(* Logix 5000 project; controller Kollmeyer_LiveDemo_TBENLX8IOL_TBIL vendor 1 type 14 code 176 rev 32.11; software revision 32.00; part 8 of 9 *)
(* IOL_WriteData, continued *)

ROUTINE Prescan   (* ladder *)
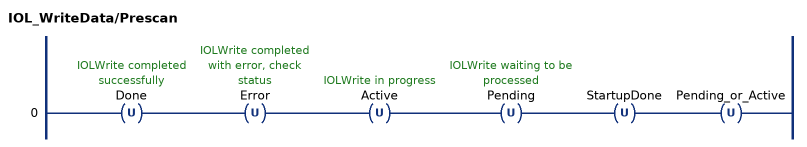
   0: OTU(Done)OTU(Error)OTU(Active)OTU(Pending)OTU(StartupDone)OTU(Pending_or_Active);
END_ROUTINE
END_ADD_ON_INSTRUCTION

ADD_ON_INSTRUCTION IOL_WriteString   (* revision 2.5 Support TBIP, ExecutePrescan, ExecuteEnableInFalse *)
// Revision note:
// V1_0 Initial Release
// V1_1 Documentation Update
// V1_3 Added multiple EIP node support
// V2_5 Support TBIP
// Help:
// IOL_WriteString - used with Turck BL20, BL67, BLC and TBEN IOLink masters to write string data to IOLink devices.  Use in conjuction with IOLService AOI which processes all IOL read and write requests.
// Status	Description
// 0	Operation completed successfully
// 	Status = 100 - 102, Ethernet IP MSG instruction errors - check communication parameters
// 100	IOL_SendMSG completed with error, check communication parameters
// 101	IOL_RecevieMSG completed with error, check communication parameters
// 110	IOL_Service Retry Limit exceeded
// 111	Slot specified not an IOLink master
// 	Status = 1000 to 1255, no response from device, connection error
// 1016	Device not connected or Port not configured as IOLink port
// 	Status = 2000 to 2255,  device response indicates error
// 2000	Device error, no details
// 2017	Device error, Index not available
// 2018	Device error, Subindex not available
// 2032	Device error, Service temporarily not available
// 2033	Device error, Service temporarily not available - local control
// 2034	Device error, Service temporarily not available - device control
// 2035	Device error, Index not writeable
// 2048	Device error, Parameter value out of range
// 2049	Device error, Parameter value above limit
// 2050	Device error, Parameter value below limit
// 2051	Device error, Parameter value length overrun (check IOLWrite precision/string length)
// 2052	Device error, Parameter value length underrun (check IOLWrite precision/string length)
// 2053	Device error, Function not available
// 2054	Device error, Function temporarily not available
// 2064	Device error, Parameter set invalid
// 2065	Device error, Inconsistent parameter set
// 2130	Device error, Application not ready
// 	Status = 3000 to 3255,   device response indicates vendor specific error
// 3000	Vendor specific error, no details
// 3001	Vendor specific error, vendor specific error number
// 3255	Vendor specific error, vendor specific error number
// 	Status = 7000 to 7255,  IOL-M Error Codes
// 7000	Unexpected write request instead of read request
// 7001	Decode error
// 7002	Port occupied by another task
// 	Status = 8000 to 8255,  IOL-M Error Codes
// 8000	Timeout when IOL-Ds or IOL-M ports are busy
// 8001	IOL Index out of range
// 8002	Port address greater than maximum
// 8003	Port function not supported
VAR_OUTPUT
   Done : BOOL; {access Read Only, visible}   // IOLWrite completed successfully
   Error : BOOL; {access Read Only, visible}   // IOLWrite completed with error, check status
   Pending : BOOL; {access Read Only, visible}   // IOLWrite waiting to be processed
   Active : BOOL; {access Read Only, visible}   // IOLWrite in progress
END_VAR
VAR_IN_OUT
   IOLData : Turck_IOL_CommonData; {required}   // Shared IOL Data Area - must be identical on all requests
END_VAR
VAR_OUTPUT
   DoneCount : DINT; {visible}   // Number of operations completed successfully
   ErrorCount : DINT; {access Read Only, visible}   // Number of operations competed with error
   Status : INT; {access Read Only, visible}   // Status of last IOLWrite
END_VAR
VAR_INPUT
   Write : BOOL;   // Rising edge triggers IOLink Write
   Slot : INT; {visible}   // IOLink Master slot number
   Port : INT; {visible}   // IOLink Master Port number, 1,2,3 or 4
   Index : INT; {visible}   // IOL Index number
   SubIndex : INT; {visible}   // IOL Subindex number
END_VAR
VAR_IN_OUT
   StringData : SINT[82]; {required}   // String data to write to IOLink device
END_VAR
VAR_INPUT
   StringLength : DINT; {access Read Only, required}   // Length of string data to write to IOLink device
END_VAR
VAR
   MyHandle : INT;
   StartupDone : BOOL; {access None}
   Pending_or_Active : BOOL; {access None}
   Write_ONS : BOOL; {access None}
   StartupCount : DINT; {access None}
   WriteRequest : BOOL; {access None}
END_VAR

ROUTINE EnableInFalse   (* ladder *)
END_ROUTINE

ROUTINE Logic   (* ladder *)
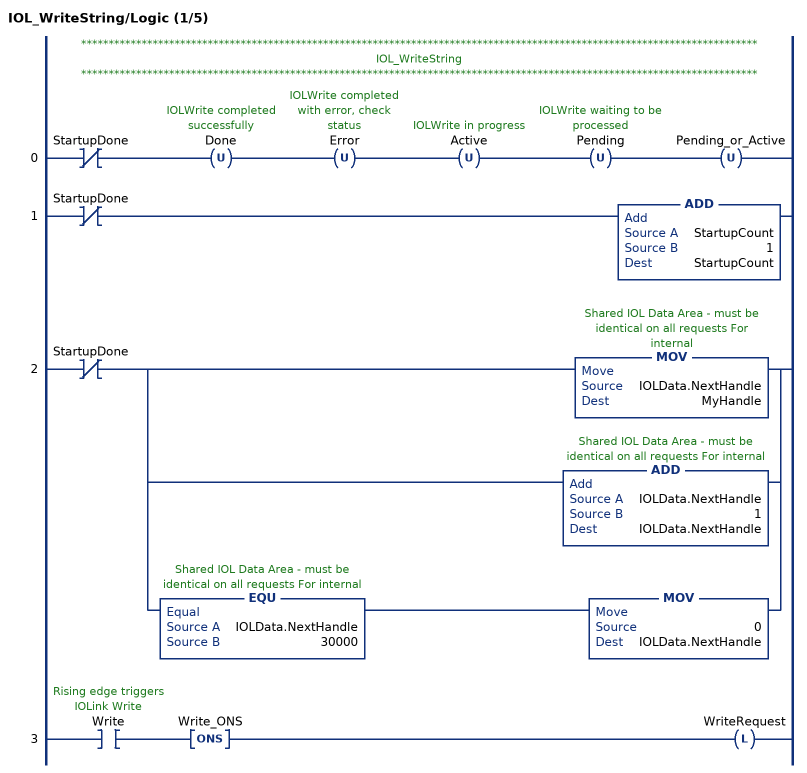
   // ***************************************************************************************************************************
   // IOL_WriteString
   // ***************************************************************************************************************************
   0: XIO(StartupDone)OTU(Done)OTU(Error)OTU(Active)OTU(Pending)OTU(Pending_or_Active);
   1: XIO(StartupDone)ADD(StartupCount,1,StartupCount);
   2: XIO(StartupDone)[MOV(IOLData.NextHandle,MyHandle) ,ADD(IOLData.NextHandle,1,IOLData.NextHandle) ,EQU(IOLData.NextHandle,30000) MOV(0,IOLData.NextHandle) ];
   3: XIC(Write)ONS(Write_ONS)OTL(WriteRequest);
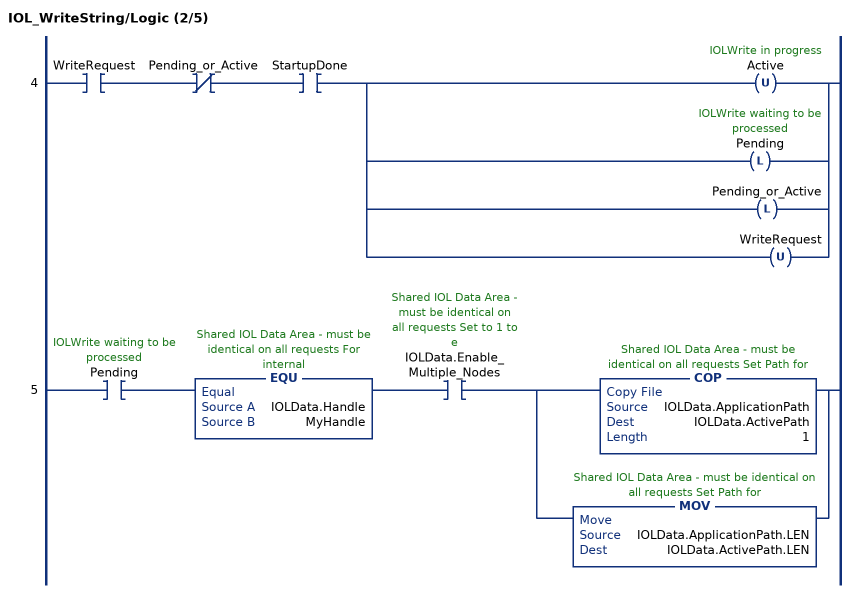
   4: XIC(WriteRequest)XIO(Pending_or_Active)XIC(StartupDone)[OTU(Active) ,OTL(Pending) ,OTL(Pending_or_Active) ,OTU(WriteRequest) ];
   5: XIC(Pending)EQU(IOLData.Handle,MyHandle)XIC(IOLData.Enable_Multiple_Nodes)[COP(IOLData.ApplicationPath,IOLData.ActivePath,1) ,MOV(IOLData.ApplicationPath.LEN,IOLData.ActivePath.LEN) ];
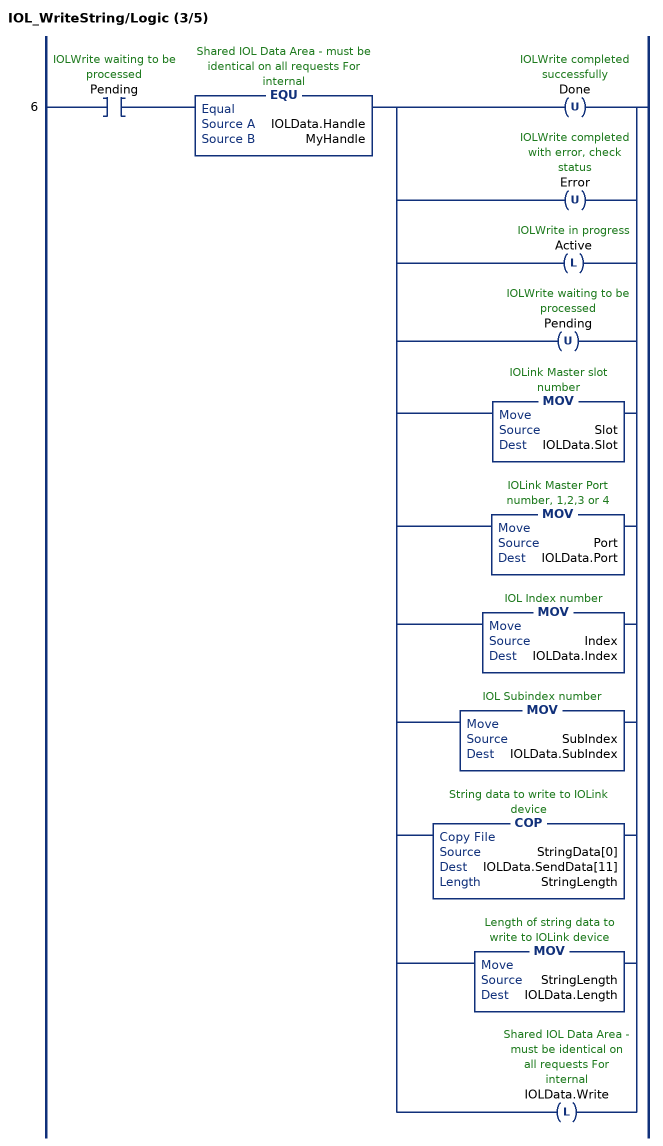
   6: XIC(Pending)EQU(IOLData.Handle,MyHandle)[OTU(Done) ,OTU(Error) ,OTL(Active) ,OTU(Pending) ,MOV(Slot,IOLData.Slot) ,MOV(Port,IOLData.Port) ,MOV(Index,IOLData.Index) ,MOV(SubIndex,IOLData.SubIndex) ,COP(StringData[0],IOLData.SendData[11],StringLength) ,MOV(StringLength,IOLData.Length) ,OTL(IOLData.Write) ];
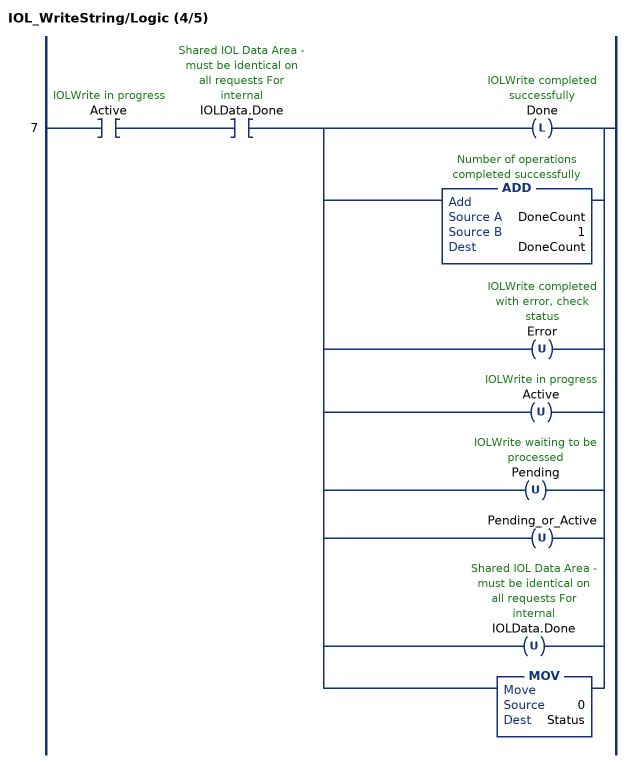
   7: XIC(Active)XIC(IOLData.Done)[OTL(Done) ,ADD(DoneCount,1,DoneCount) ,OTU(Error) ,OTU(Active) ,OTU(Pending) ,OTU(Pending_or_Active) ,OTU(IOLData.Done) ,MOV(0,Status) ];
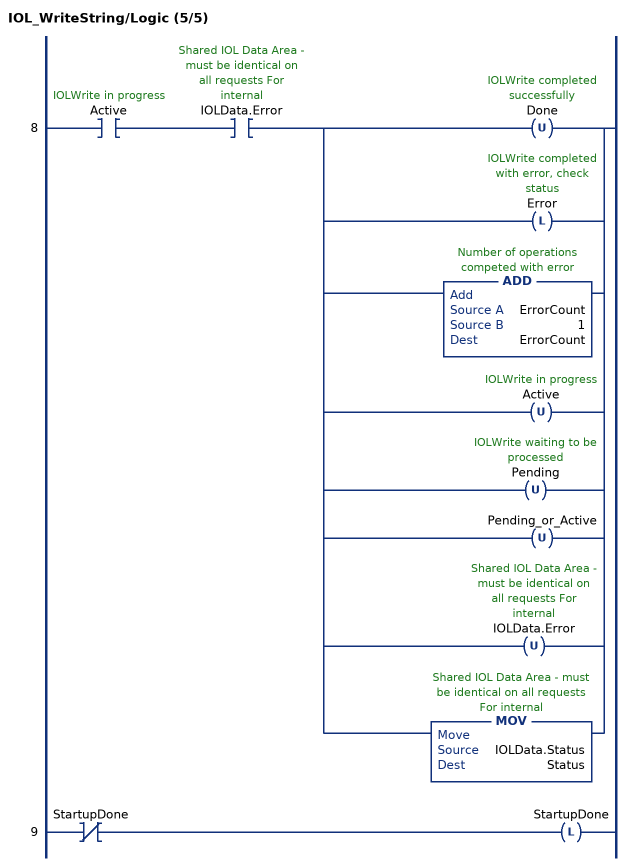
   8: XIC(Active)XIC(IOLData.Error)[OTU(Done) ,OTL(Error) ,ADD(ErrorCount,1,ErrorCount) ,OTU(Active) ,OTU(Pending) ,OTU(Pending_or_Active) ,OTU(IOLData.Error) ,MOV(IOLData.Status,Status) ];
   9: XIO(StartupDone)OTL(StartupDone);
END_ROUTINE

ROUTINE Prescan   (* ladder *)
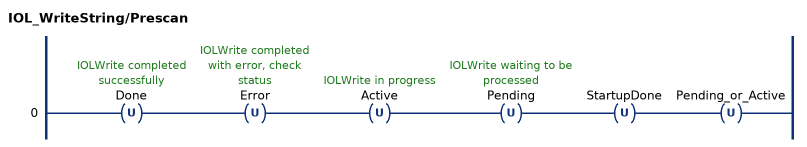
   0: OTU(Done)OTU(Error)OTU(Active)OTU(Pending)OTU(StartupDone)OTU(Pending_or_Active);
END_ROUTINE
END_ADD_ON_INSTRUCTION

ADD_ON_INSTRUCTION TBEN_L_8IOL_AOI   (* revision 0.1 Support TBIP, ExecutePrescan *)
// TBEN_L_8IOL AOI for managing all data to/from IOL blocks including process/acyclic data.
// Revision note:
// V0_1 Testing
// Help:
// IOL_Service - used with Turck BL20, BL67, BLC and TBEN IOLink masters to process requests from IOL_ReadString, IOL_WriteString, IOL_ReadData and IOL_WriteData AOI's.
// Status	Description
// 0	Operation completed successfully
// 	Status = 100 - 102, Ethernet IP MSG instruction errors - check communication parameters
// 100	IOL_SendMSG completed with error, check communication parameters
// 101	IOL_RecevieMSG completed with error, check communication parameters
// 110	IOL_Service Retry Limit exceeded
// 111	Slot specified not an IOLink master
// 	Status = 1000 to 1255, no response from device, connection error
// 1016	Device not connected or Port not configured as IOLink port
// 	Status = 2000 to 2255,  device response indicates error
// 2000	Device error, no details
// 2017	Device error, Index not available
// 2018	Device error, Subindex not available
// 2032	Device error, Service temporarily not available
// 2033	Device error, Service temporarily not available - local control
// 2034	Device error, Service temporarily not available - device control
// 2035	Device error, Index not writeable
// 2048	Device error, Parameter value out of range
// 2049	Device error, Parameter value above limit
// 2050	Device error, Parameter value below limit
// 2051	Device error, Parameter value length overrun (check IOLWrite precision/string length)
// 2052	Device error, Parameter value length underrun (check IOLWrite precision/string length)
// 2053	Device error, Function not available
// 2054	Device error, Function temporarily not available
// 2064	Device error, Parameter set invalid
// 2065	Device error, Inconsistent parameter set
// 2130	Device error, Application not ready
// 	Status = 3000 to 3255,   device response indicates vendor specific error
// 3000	Vendor specific error, no details
// 3001	Vendor specific error, vendor specific error number
// 3255	Vendor specific error, vendor specific error number
// 	Status = 7000 to 7255,  IOL-M Error Codes
// 7000	Unexpected write request instead of read request
// 7001	Decode error
// 7002	Port occupied by another task
// 	Status = 8000 to 8255,  IOL-M Error Codes
// 8000	Timeout when IOL-Ds or IOL-M ports are busy
// 8001	IOL Index out of range
// 8002	Port address greater than maximum
// 8003	Port function not supported
VAR_IN_OUT
   Process_Input_Data : Generic_173_Words; {required}
   Process_Output_Data : Generic_131_Words; {required}
   CommonData : Turck_IOL_CommonData; {required}
        .ReceiveData[2]   // KH changed from -9 (f7) to -4 (Fd)
        .SendData[1]   // For internal use to integrate IOLRead and IOLWrite with IOLService
   IOL_SendMSG : MESSAGE; {required}
   IOL_ReceiveMSG : MESSAGE; {required}
END_VAR
VAR_OUTPUT
   Port1_VID : DINT; {visible}
   Port1_DID : DINT; {visible}
   Port2_VID : DINT; {visible}
   Port2_DID : DINT; {visible}
   Port3_VID : DINT; {visible}
   Port3_DID : DINT; {visible}
   Port4_VID : DINT; {visible}
   Port4_DID : DINT; {visible}
   Port5_VID : DINT; {visible}
   Port5_DID : DINT; {visible}
   Port6_VID : DINT; {visible}
   Port6_DID : DINT; {visible}
   Port7_VID : DINT; {visible}
   Port7_DID : DINT; {visible}
   Port8_VID : DINT; {visible}
   Port8_DID : DINT; {visible}
   Port1_SN : DINT; {access Read Only}
   Port1_COMRev : DINT;
   Port1_ProcInLenght : DINT;
   Port1_ProcOutLenght : DINT;
   Port1_CycleTime : DINT;
   Port2_SN : DINT;
   Port2_COMRev : DINT;
   Port2_ProcInLenght : DINT;
   Port2_ProcOutLenght : DINT;
   Port2_CycleTime : DINT;
   Port3_SN : DINT;
   Port3_COMRev : DINT;
   Port3_ProcInLenght : DINT;
   Port3_ProcOutLenght : DINT;
   Port3_CycleTime : DINT;
   Port4_SN : DINT;
   Port4_COMRev : DINT;
   Port4_ProcInLenght : DINT;
   Port4_ProcOutLenght : DINT;
   Port4_CycleTime : DINT;
   Port5_SN : DINT;
   Port5_COMRev : DINT;
   Port5_ProcInLenght : DINT;
   Port5_ProcOutLenght : DINT;
   Port5_CycleTime : DINT;
   Port6_SN : DINT;
   Port6_COMRev : DINT;
   Port6_ProcInLenght : DINT;
   Port6_ProcOutLenght : DINT;
   Port6_CycleTime : DINT;
   Port7_SN : DINT;
   Port7_COMRev : DINT;
   Port7_ProcInLenght : DINT;
   Port7_ProcOutLenght : DINT;
   Port7_CycleTime : DINT;
   Port8_SN : DINT;
   Port8_COMRev : DINT;
   Port8_ProcInLenght : DINT;
   Port8_ProcOutLenght : DINT;
   Port8_CycleTime : DINT;
END_VAR
VAR
   IOLS1 : BOOL;
   IOLS2 : BOOL;
   IOLS3 : BOOL;
   IOLS4 : BOOL;
   IOLS5 : BOOL;
   IOLS6 : BOOL;
   IOLS7 : BOOL;
   IOLReadActive : BOOL;
   IOLWriteActive : BOOL;
   Retry : BOOL;
   RetryCount : DINT;
   IOL_SendMSG_Request : BOOL; {access None}
   IOL_ReceiveMSG_Request : BOOL; {access None}
   IOLS4_Bad : BOOL; {access None}
   IOL_S2_0_Count : DINT; {access None}
   IOL_S6_0_Count : DINT; {access None}
   Busy_Retry : BOOL; {access None}
   IOL_S2_0_Total : DINT; {access None}
   IOL_S3_Retry : DINT; {access None}
   IOL_S1_Count : DINT; {access None}
   IOL_S2_Count : DINT; {access None}
   IOL_S3_Count : DINT; {access None}
   IOL_S5_Count : DINT; {access None}
   IOL_S6_Count : DINT; {access None}
   ER1 : BOOL; {access None}
   ER2 : BOOL; {access None}
   IOL_S6_NotBusy_Count : DINT; {access None}
   RetryTotal : DINT; {access None}
   IOL_S4_Bad_Count : DINT; {access None}
   IOL_S2_Error_Count : DINT; {access None}
   IOL_Done_Count : DINT; {access None}
   IOL_Error_Count : DINT; {access None}
   IOLReset_ONS : BOOL; {access None}
   ABS_RD_11 : INT; {access None}
   ABS_RD_12 : INT; {access None}
   ABS_RD_13 : INT; {access None}
   IOL_SendMSG_DN : BOOL; {access None}
   IOL_ReceiveMSG_DN : BOOL; {access None}
   IOLS2A : BOOL; {access None}
   Generate_Status : BOOL; {access None}
   IOLS5A : BOOL; {access None}
   Busy_Response : BOOL; {access None}
   Done_Response : BOOL; {access None}
   IOL_S6_Done_Count : DINT; {access None}
   Wait : BOOL; {access None}
   IOL_S6_Busy_Count : DINT; {access None}
   PORT_DATA : SINT[230]; {access None}
   PORT_DATA_LENGHT : DINT; {access None}
   READ_PORT_DATA : IOL_ReadString := (Slot := 1, Index := -1, SubIndex := 68); {access None}
END_VAR

ROUTINE Logic   (* ladder *)
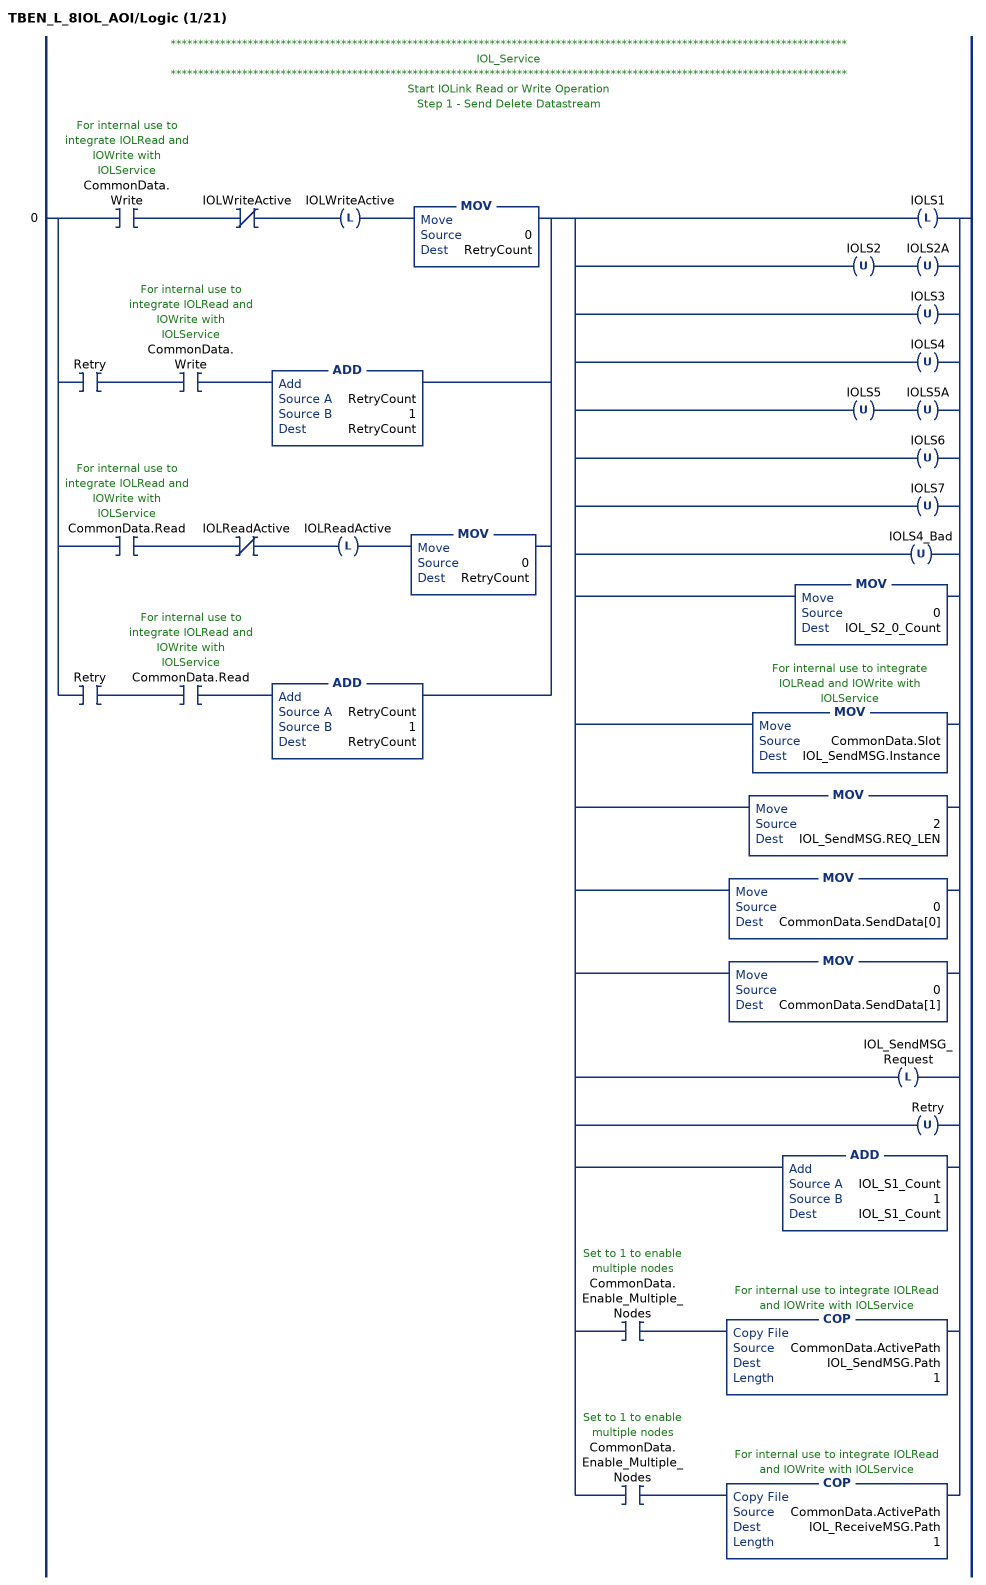
   // ***************************************************************************************************************************
   // IOL_Service
   // ***************************************************************************************************************************
   // Start IOLink Read or Write Operation
   // Step 1 - Send Delete Datastream
   0: [XIC(CommonData.Write) XIO(IOLWriteActive) OTL(IOLWriteActive) MOV(0,RetryCount) ,XIC(Retry) XIC(CommonData.Write) ADD(RetryCount,1,RetryCount) ,XIC(CommonData.Read) XIO(IOLReadActive) OTL(IOLReadActive) MOV(0,RetryCount) ,XIC(Retry) XIC(CommonData.Read) ADD(RetryCount,1,RetryCount) ][OTL(IOLS1) ,OTU(IOLS2) OTU(IOLS2A) ,OTU(IOLS3) ,OTU(IOLS4) ,OTU(IOLS5) OTU(IOLS5A) ,OTU(IOLS6) ,OTU(IOLS7) ,OTU(IOLS4_Bad) ,MOV(0,IOL_S2_0_Count) ,MOV(CommonData.Slot,IOL_SendMSG.Instance) ,MOV(2,IOL_SendMSG.REQ_LEN) ,MOV(0,CommonData.SendData[0]) ,MOV(0,CommonData.SendData[1]) ,OTL(IOL_SendMSG_Request) ,OTU(Retry) ,ADD(IOL_S1_Count,1,IOL_S1_Count) ,XIC(CommonData.Enable_Multiple_Nodes) COP(CommonData.ActivePath,IOL_SendMSG.Path,1) ,XIC(CommonData.Enable_Multiple_Nodes) COP(CommonData.ActivePath,IOL_ReceiveMSG.Path,1) ];
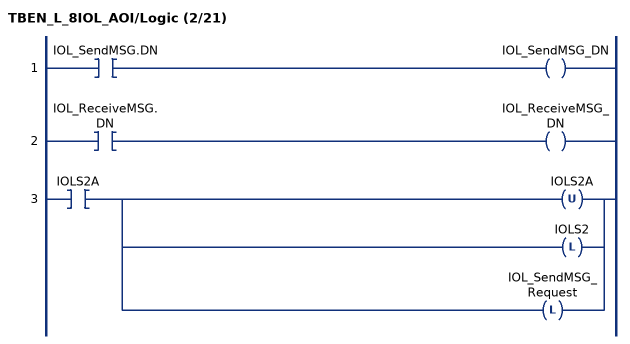
   1: XIC(IOL_SendMSG.DN)OTE(IOL_SendMSG_DN);
   2: XIC(IOL_ReceiveMSG.DN)OTE(IOL_ReceiveMSG_DN);
   3: XIC(IOLS2A)[OTU(IOLS2A) ,OTL(IOLS2) ,OTL(IOL_SendMSG_Request) ];
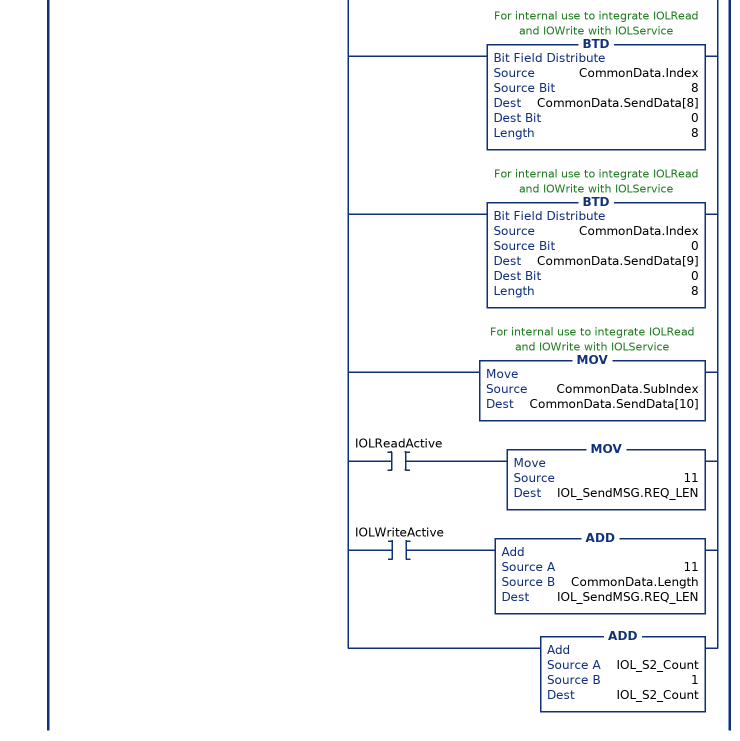
   // Step 1 - After Delete Stream sent then Send IOLink Read or Write Request
   4: XIC(IOLS1)XIC(IOL_SendMSG_DN)XIO(IOL_SendMSG_Request)[OTU(IOLS1) ,OTL(IOLS2A) ,MOV(CommonData.Slot,IOL_SendMSG.Instance) ,MOV(0,CommonData.SendData[0]) ,MOV(16#fc,CommonData.SendData[1]) ,MOV(16#11,CommonData.SendData[2]) ,MOV(16#08,CommonData.SendData[3]) ,MOV(CommonData.Port,CommonData.SendData[4]) ,MOV(16#fe,CommonData.SendData[5]) ,MOV(16#4a,CommonData.SendData[6]) ,XIC(IOLReadActive) MOV(16#03,CommonData.SendData[7]) ,XIC(IOLWriteActive) MOV(16#02,CommonData.SendData[7]) ,BTD(CommonData.Index,8,CommonData.SendData[8],0,8) ,BTD(CommonData.Index,0,CommonData.SendData[9],0,8) ,MOV(CommonData.SubIndex,CommonData.SendData[10]) ,XIC(IOLReadActive) MOV(11,IOL_SendMSG.REQ_LEN) ,XIC(IOLWriteActive) ADD(11,CommonData.Length,IOL_SendMSG.REQ_LEN) ,ADD(IOL_S2_Count,1,IOL_S2_Count) ];
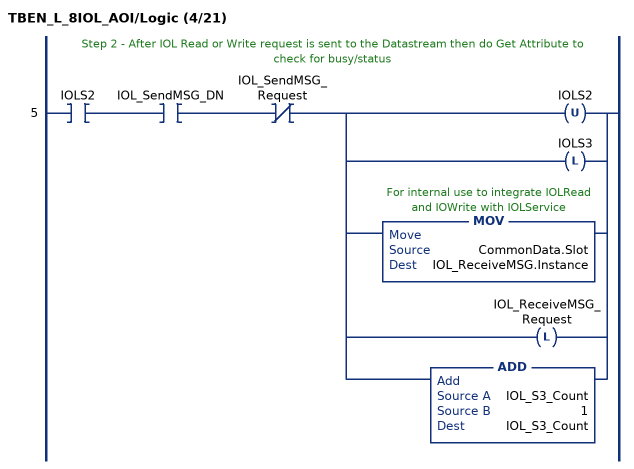
   // Step 2 - After IOL Read or Write request is sent to the Datastream then do Get Attribute to check for busy/status
   5: XIC(IOLS2)XIC(IOL_SendMSG_DN)XIO(IOL_SendMSG_Request)[OTU(IOLS2) ,OTL(IOLS3) ,MOV(CommonData.Slot,IOL_ReceiveMSG.Instance) ,OTL(IOL_ReceiveMSG_Request) ,ADD(IOL_S3_Count,1,IOL_S3_Count) ];
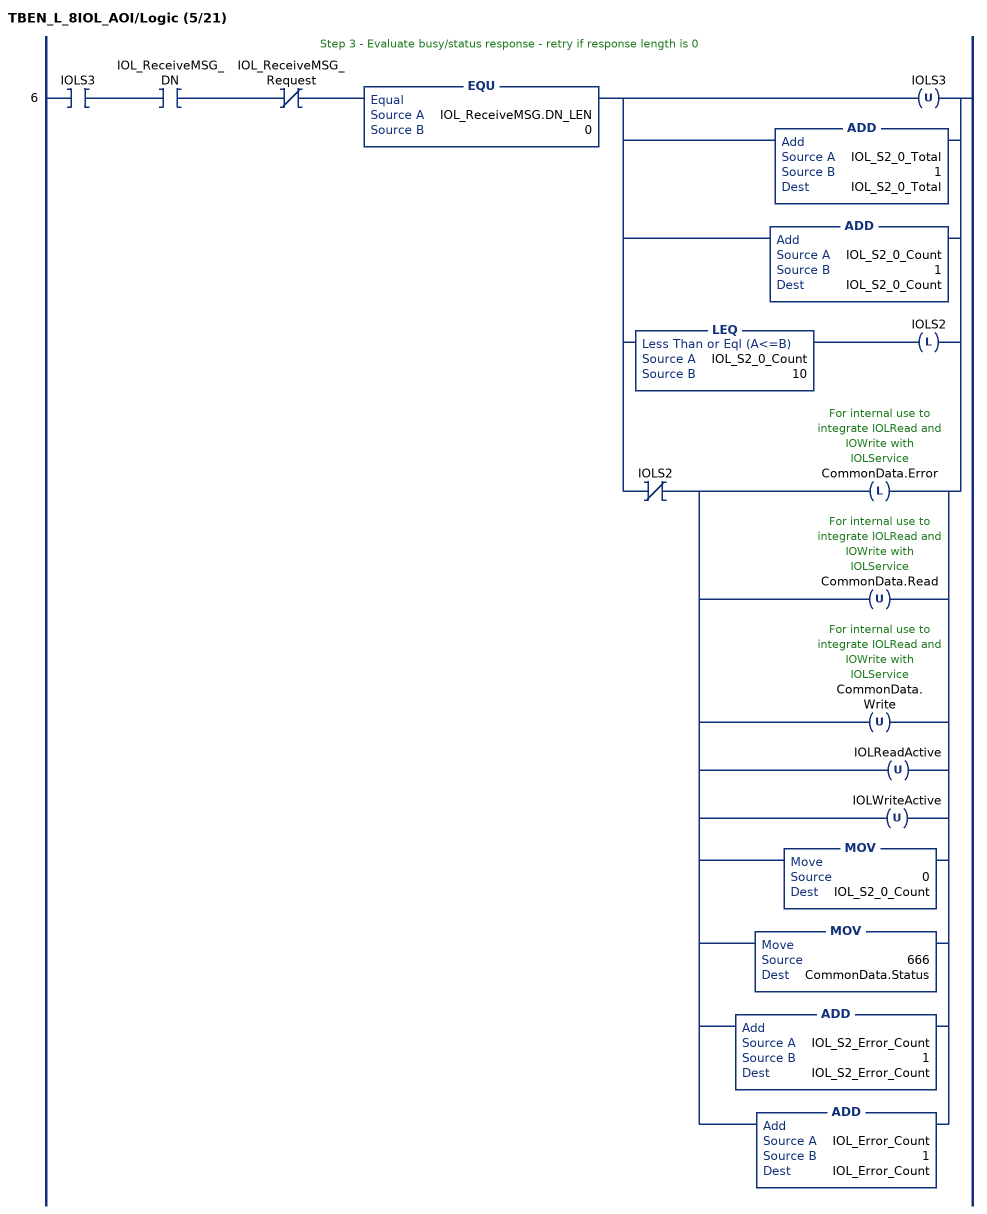
   // Step 3 - Evaluate busy/status response - retry if response length is 0
   6: XIC(IOLS3)XIC(IOL_ReceiveMSG_DN)XIO(IOL_ReceiveMSG_Request)EQU(IOL_ReceiveMSG.DN_LEN,0)[OTU(IOLS3) ,ADD(IOL_S2_0_Total,1,IOL_S2_0_Total) ,ADD(IOL_S2_0_Count,1,IOL_S2_0_Count) ,LEQ(IOL_S2_0_Count,10) OTL(IOLS2) ,XIO(IOLS2) [OTL(CommonData.Error) ,OTU(CommonData.Read) ,OTU(CommonData.Write) ,OTU(IOLReadActive) ,OTU(IOLWriteActive) ,MOV(0,IOL_S2_0_Count) ,MOV(666,CommonData.Status) ,ADD(IOL_S2_Error_Count,1,IOL_S2_Error_Count) ,ADD(IOL_Error_Count,1,IOL_Error_Count) ] ];
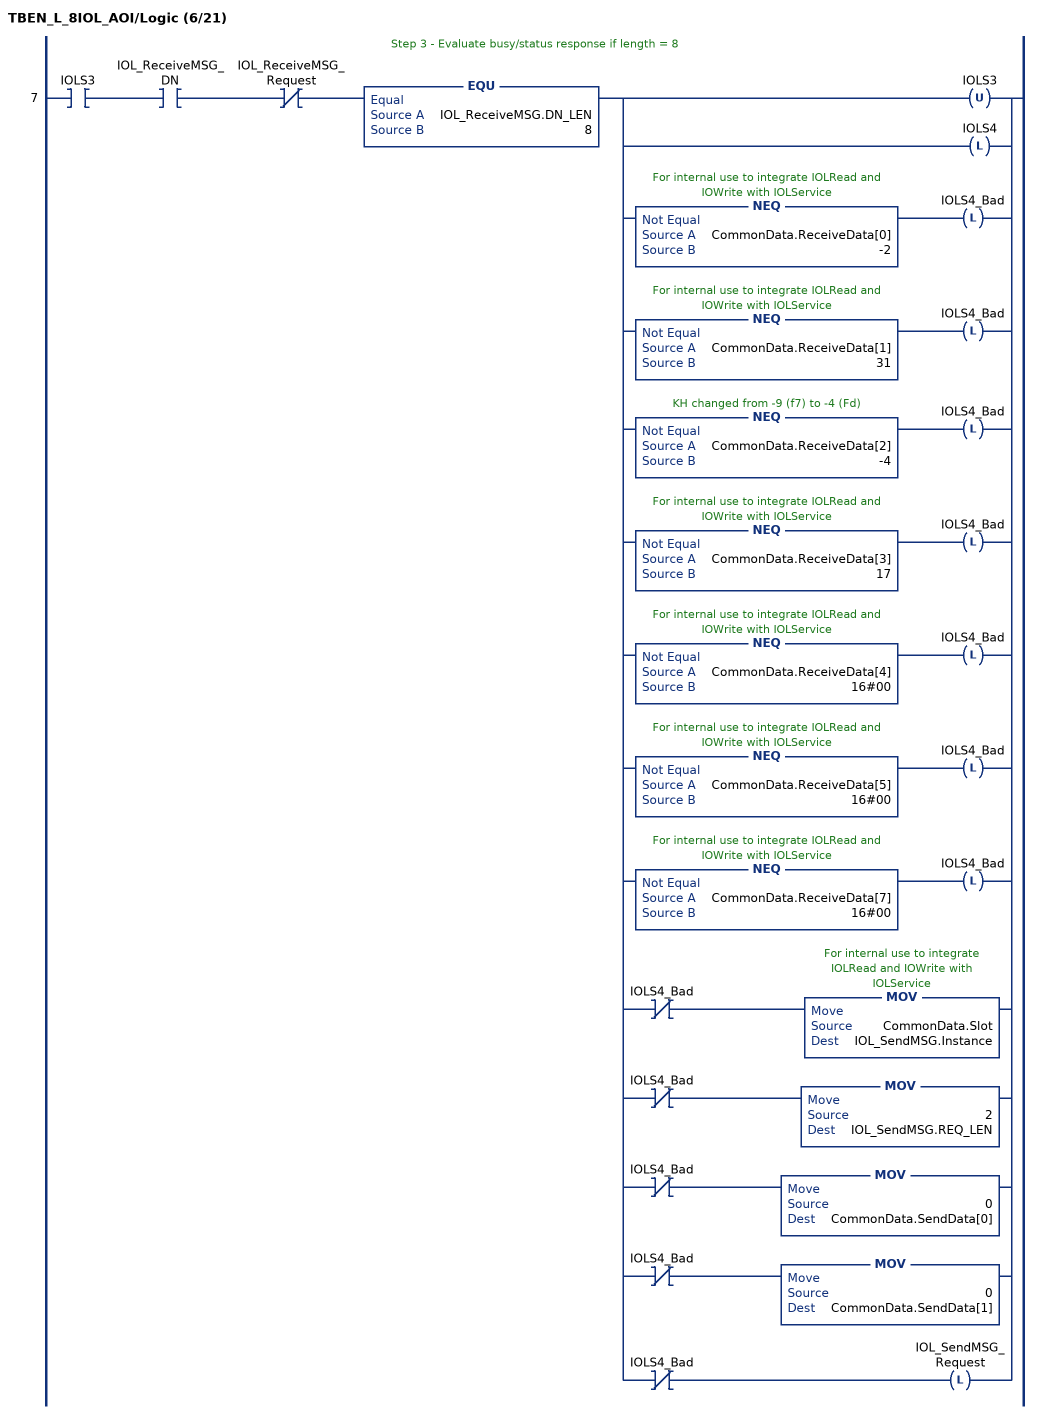
   // Step 3 - Evaluate busy/status response if length = 8
   7: XIC(IOLS3)XIC(IOL_ReceiveMSG_DN)XIO(IOL_ReceiveMSG_Request)EQU(IOL_ReceiveMSG.DN_LEN,8)[OTU(IOLS3) ,OTL(IOLS4) ,NEQ(CommonData.ReceiveData[0],-2) OTL(IOLS4_Bad) ,NEQ(CommonData.ReceiveData[1],31) OTL(IOLS4_Bad) ,NEQ(CommonData.ReceiveData[2],-4) OTL(IOLS4_Bad) ,NEQ(CommonData.ReceiveData[3],17) OTL(IOLS4_Bad) ,NEQ(CommonData.ReceiveData[4],16#00) OTL(IOLS4_Bad) ,NEQ(CommonData.ReceiveData[5],16#00) OTL(IOLS4_Bad) ,NEQ(CommonData.ReceiveData[7],16#00) OTL(IOLS4_Bad) ,XIO(IOLS4_Bad) MOV(CommonData.Slot,IOL_SendMSG.Instance) ,XIO(IOLS4_Bad) MOV(2,IOL_SendMSG.REQ_LEN) ,XIO(IOLS4_Bad) MOV(0,CommonData.SendData[0]) ,XIO(IOLS4_Bad) MOV(0,CommonData.SendData[1]) ,XIO(IOLS4_Bad) OTL(IOL_SendMSG_Request) ];
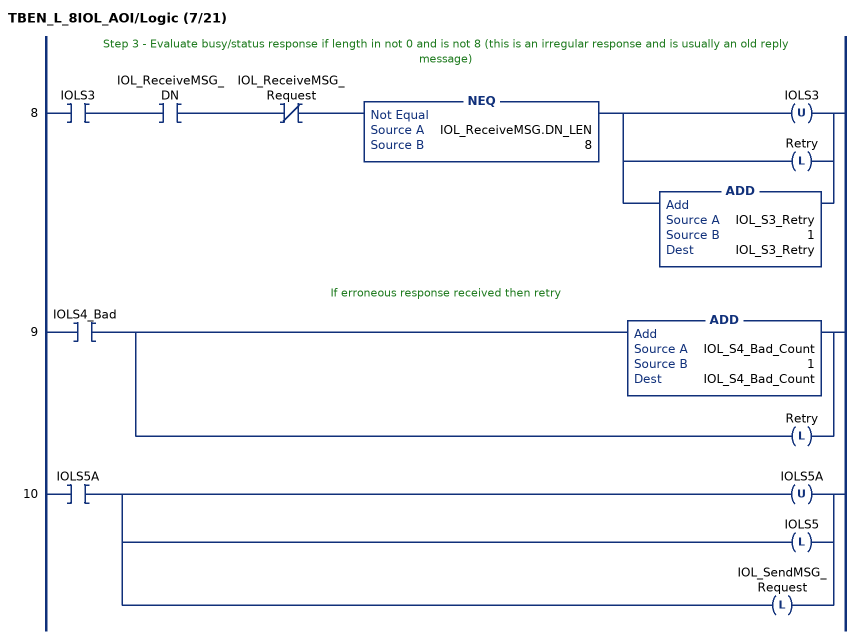
   // Step 3 - Evaluate busy/status response if length in not 0 and is not 8 (this is an irregular response and is usually an old reply message)
   8: XIC(IOLS3)XIC(IOL_ReceiveMSG_DN)XIO(IOL_ReceiveMSG_Request)NEQ(IOL_ReceiveMSG.DN_LEN,8)[OTU(IOLS3) ,OTL(Retry) ,ADD(IOL_S3_Retry,1,IOL_S3_Retry) ];
   // If erroneous response received then retry
   9: XIC(IOLS4_Bad)[ADD(IOL_S4_Bad_Count,1,IOL_S4_Bad_Count) ,OTL(Retry) ];
   10: XIC(IOLS5A)[OTU(IOLS5A) ,OTL(IOLS5) ,OTL(IOL_SendMSG_Request) ];
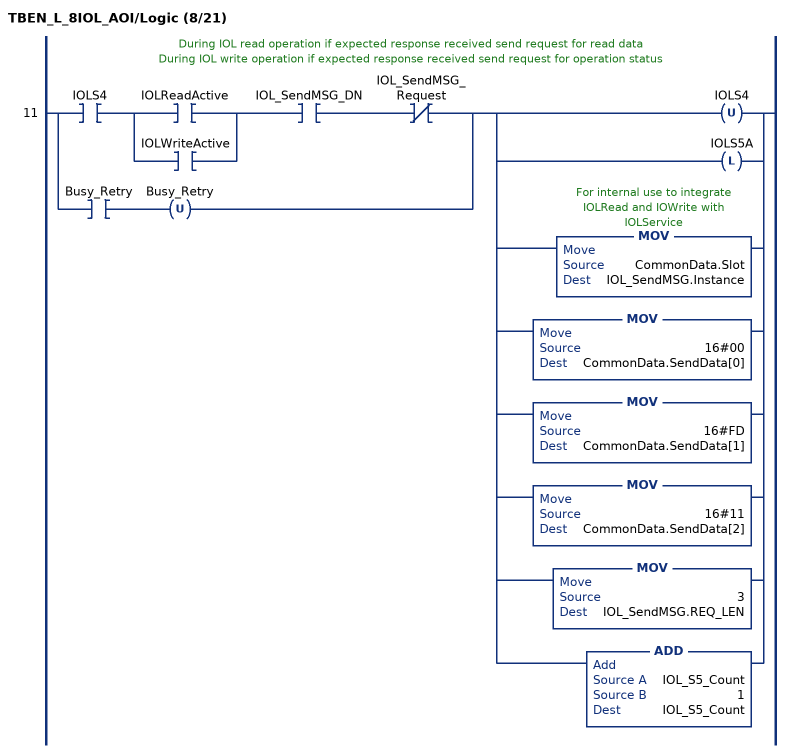
   // During IOL read operation if expected response received send request for read data
   // During IOL write operation if expected response received send request for operation status
   11: [XIC(IOLS4) [XIC(IOLReadActive) ,XIC(IOLWriteActive) ] XIC(IOL_SendMSG_DN) XIO(IOL_SendMSG_Request) ,XIC(Busy_Retry) OTU(Busy_Retry) ][OTU(IOLS4) ,OTL(IOLS5A) ,MOV(CommonData.Slot,IOL_SendMSG.Instance) ,MOV(16#00,CommonData.SendData[0]) ,MOV(16#FD,CommonData.SendData[1]) ,MOV(16#11,CommonData.SendData[2]) ,MOV(3,IOL_SendMSG.REQ_LEN) ,ADD(IOL_S5_Count,1,IOL_S5_Count) ];
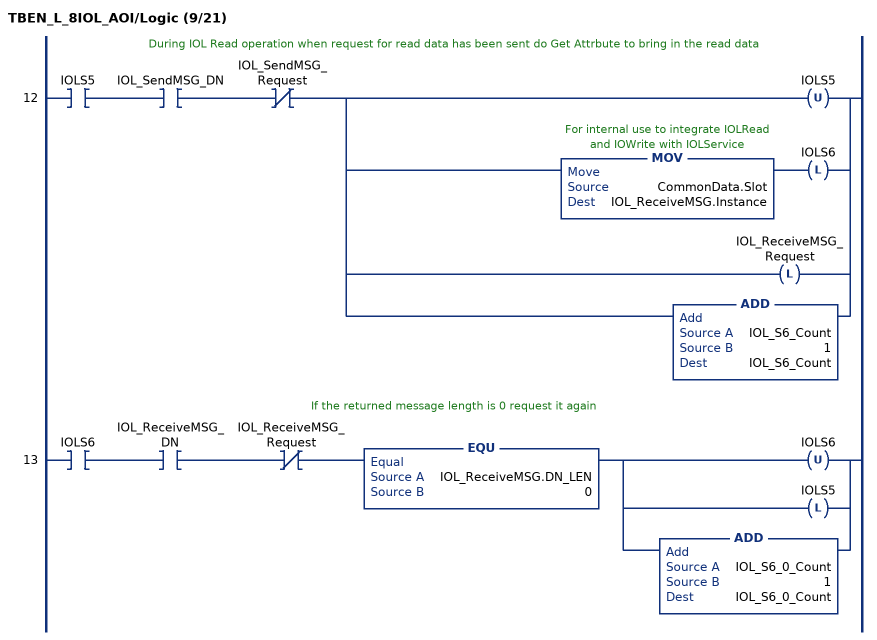
   // During IOL Read operation when request for read data has been sent do Get Attrbute to bring in the read data
   12: XIC(IOLS5)XIC(IOL_SendMSG_DN)XIO(IOL_SendMSG_Request)[OTU(IOLS5) ,MOV(CommonData.Slot,IOL_ReceiveMSG.Instance) OTL(IOLS6) ,OTL(IOL_ReceiveMSG_Request) ,ADD(IOL_S6_Count,1,IOL_S6_Count) ];
   // If the returned message length is 0 request it again
   13: XIC(IOLS6)XIC(IOL_ReceiveMSG_DN)XIO(IOL_ReceiveMSG_Request)EQU(IOL_ReceiveMSG.DN_LEN,0)[OTU(IOLS6) ,OTL(IOLS5) ,ADD(IOL_S6_0_Count,1,IOL_S6_0_Count) ];
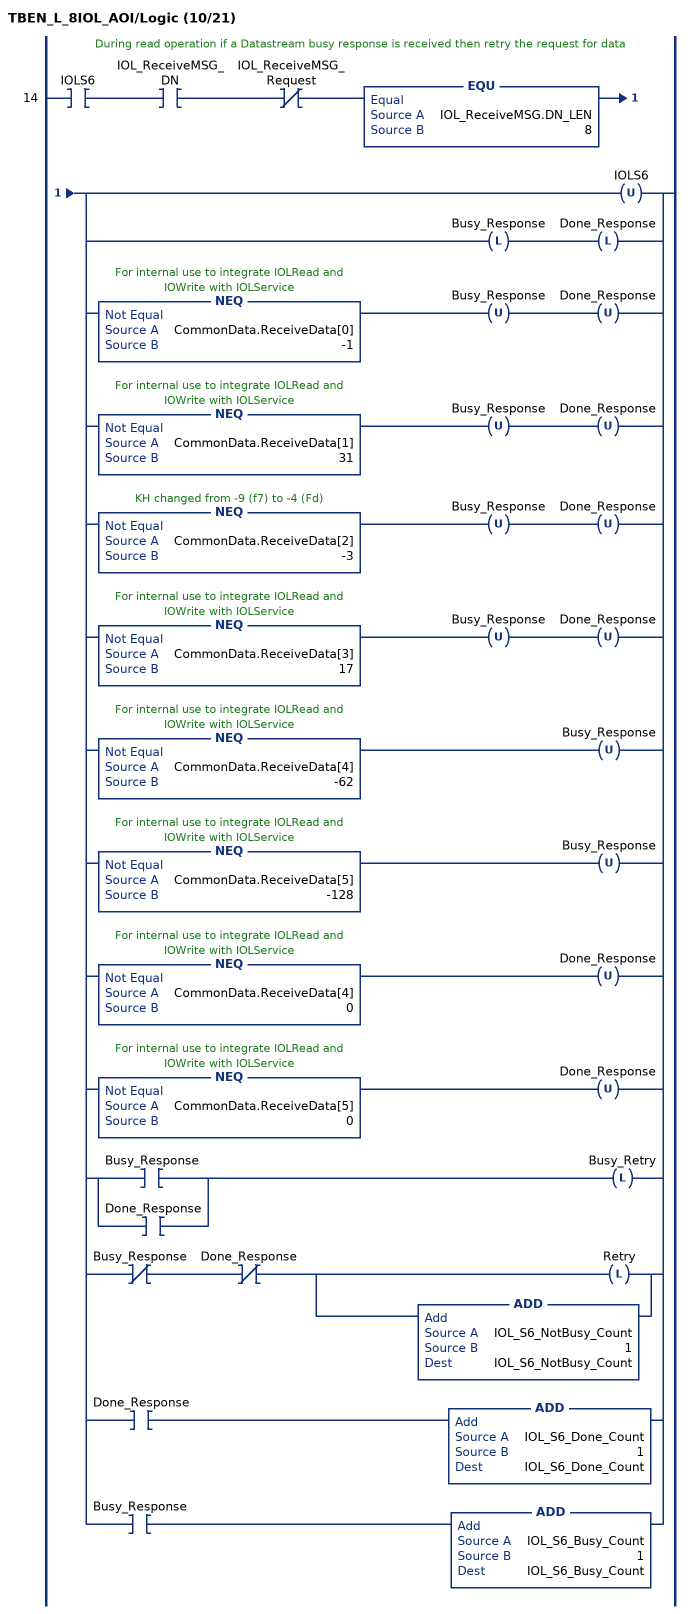
   // During read operation if a Datastream busy response is received then retry the request for data
   14: XIC(IOLS6)XIC(IOL_ReceiveMSG_DN)XIO(IOL_ReceiveMSG_Request)EQU(IOL_ReceiveMSG.DN_LEN,8)[OTU(IOLS6) ,OTL(Busy_Response) OTL(Done_Response) ,NEQ(CommonData.ReceiveData[0],-1) OTU(Busy_Response) OTU(Done_Response) ,NEQ(CommonData.ReceiveData[1],31) OTU(Busy_Response) OTU(Done_Response) ,NEQ(CommonData.ReceiveData[2],-3) OTU(Busy_Response) OTU(Done_Response) ,NEQ(CommonData.ReceiveData[3],17) OTU(Busy_Response) OTU(Done_Response) ,NEQ(CommonData.ReceiveData[4],-62) OTU(Busy_Response) ,NEQ(CommonData.ReceiveData[5],-128) OTU(Busy_Response) ,NEQ(CommonData.ReceiveData[4],0) OTU(Done_Response) ,NEQ(CommonData.ReceiveData[5],0) OTU(Done_Response) ,[XIC(Busy_Response) ,XIC(Done_Response) ] OTL(Busy_Retry) ,XIO(Busy_Response) XIO(Done_Response) [OTL(Retry) ,ADD(IOL_S6_NotBusy_Count,1,IOL_S6_NotBusy_Count) ] ,XIC(Done_Response) ADD(IOL_S6_Done_Count,1,IOL_S6_Done_Count) ,XIC(Busy_Response) ADD(IOL_S6_Busy_Count,1,IOL_S6_Busy_Count) ];
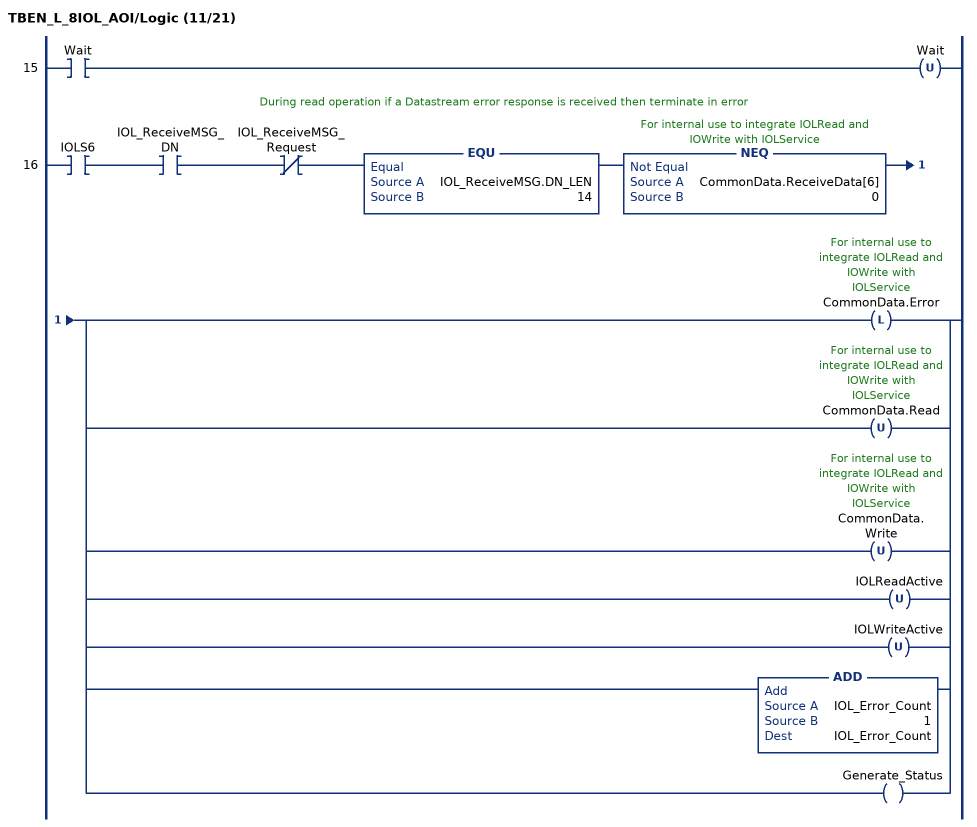
   15: XIC(Wait)OTU(Wait);
   // During read operation if a Datastream error response is received then terminate in error
   16: XIC(IOLS6)XIC(IOL_ReceiveMSG_DN)XIO(IOL_ReceiveMSG_Request)EQU(IOL_ReceiveMSG.DN_LEN,14)NEQ(CommonData.ReceiveData[6],0)[OTL(CommonData.Error) ,OTU(CommonData.Read) ,OTU(CommonData.Write) ,OTU(IOLReadActive) ,OTU(IOLWriteActive) ,ADD(IOL_Error_Count,1,IOL_Error_Count) ,OTE(Generate_Status) ];
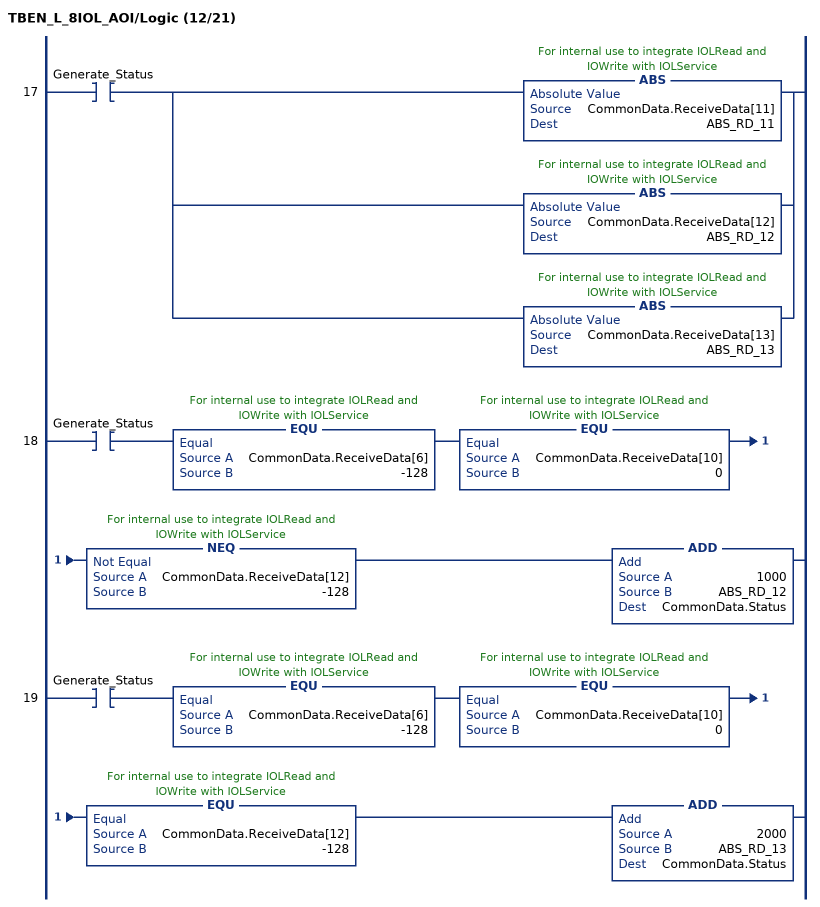
   17: XIC(Generate_Status)[ABS(CommonData.ReceiveData[11],ABS_RD_11) ,ABS(CommonData.ReceiveData[12],ABS_RD_12) ,ABS(CommonData.ReceiveData[13],ABS_RD_13) ];
   18: XIC(Generate_Status)EQU(CommonData.ReceiveData[6],-128)EQU(CommonData.ReceiveData[10],0)NEQ(CommonData.ReceiveData[12],-128)ADD(1000,ABS_RD_12,CommonData.Status);
   19: XIC(Generate_Status)EQU(CommonData.ReceiveData[6],-128)EQU(CommonData.ReceiveData[10],0)EQU(CommonData.ReceiveData[12],-128)ADD(2000,ABS_RD_13,CommonData.Status);
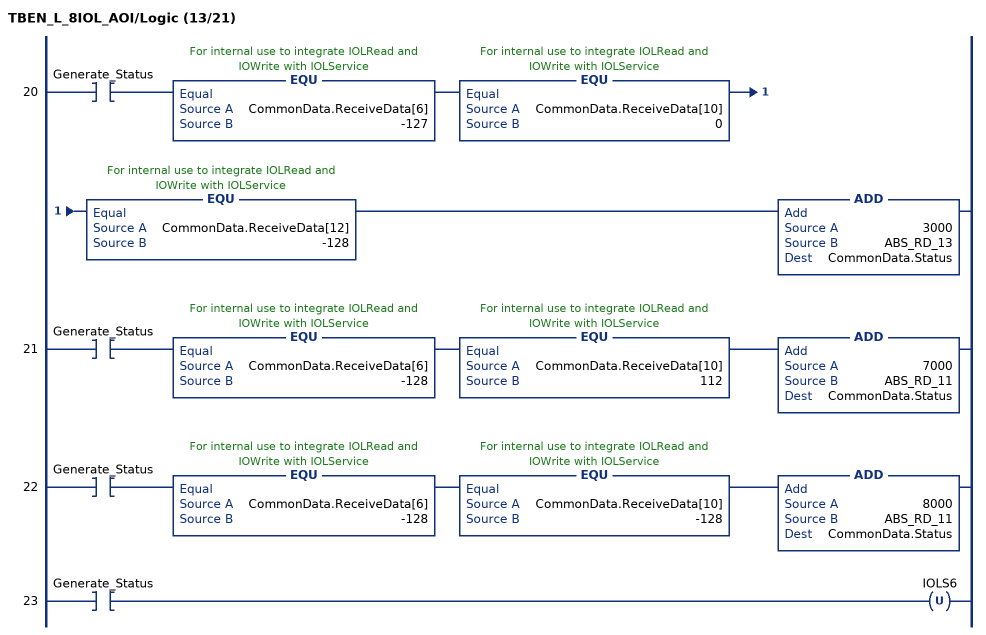
   20: XIC(Generate_Status)EQU(CommonData.ReceiveData[6],-127)EQU(CommonData.ReceiveData[10],0)EQU(CommonData.ReceiveData[12],-128)ADD(3000,ABS_RD_13,CommonData.Status);
   21: XIC(Generate_Status)EQU(CommonData.ReceiveData[6],-128)EQU(CommonData.ReceiveData[10],112)ADD(7000,ABS_RD_11,CommonData.Status);
   22: XIC(Generate_Status)EQU(CommonData.ReceiveData[6],-128)EQU(CommonData.ReceiveData[10],-128)ADD(8000,ABS_RD_11,CommonData.Status);
   23: XIC(Generate_Status)OTU(IOLS6);
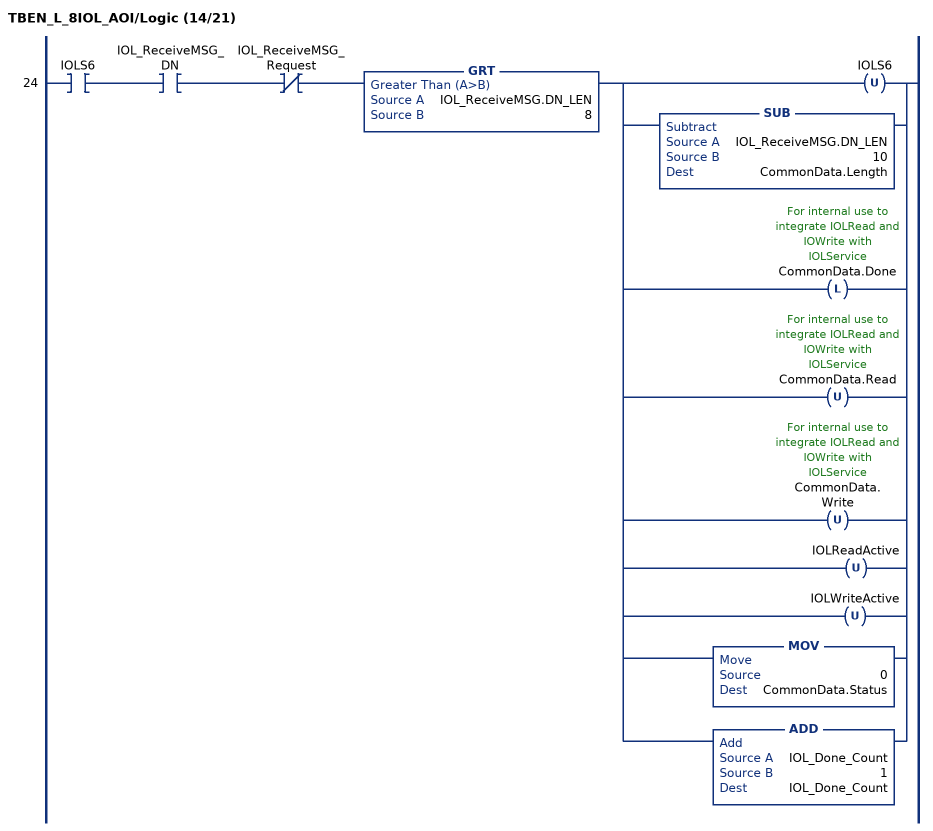
   24: XIC(IOLS6)XIC(IOL_ReceiveMSG_DN)XIO(IOL_ReceiveMSG_Request)GRT(IOL_ReceiveMSG.DN_LEN,8)[OTU(IOLS6) ,SUB(IOL_ReceiveMSG.DN_LEN,10,CommonData.Length) ,OTL(CommonData.Done) ,OTU(CommonData.Read) ,OTU(CommonData.Write) ,OTU(IOLReadActive) ,OTU(IOLWriteActive) ,MOV(0,CommonData.Status) ,ADD(IOL_Done_Count,1,IOL_Done_Count) ];
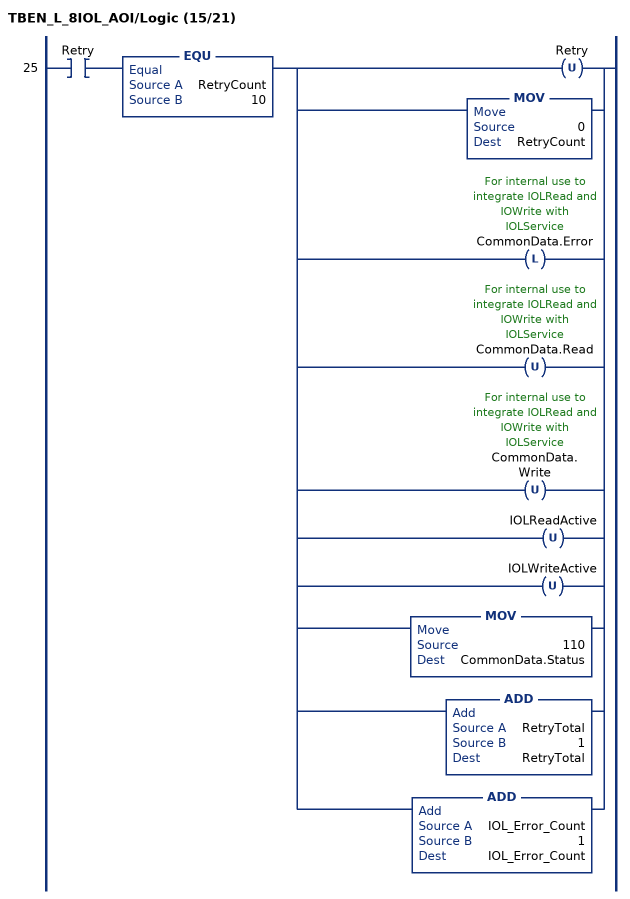
   25: XIC(Retry)EQU(RetryCount,10)[OTU(Retry) ,MOV(0,RetryCount) ,OTL(CommonData.Error) ,OTU(CommonData.Read) ,OTU(CommonData.Write) ,OTU(IOLReadActive) ,OTU(IOLWriteActive) ,MOV(110,CommonData.Status) ,ADD(RetryTotal,1,RetryTotal) ,ADD(IOL_Error_Count,1,IOL_Error_Count) ];
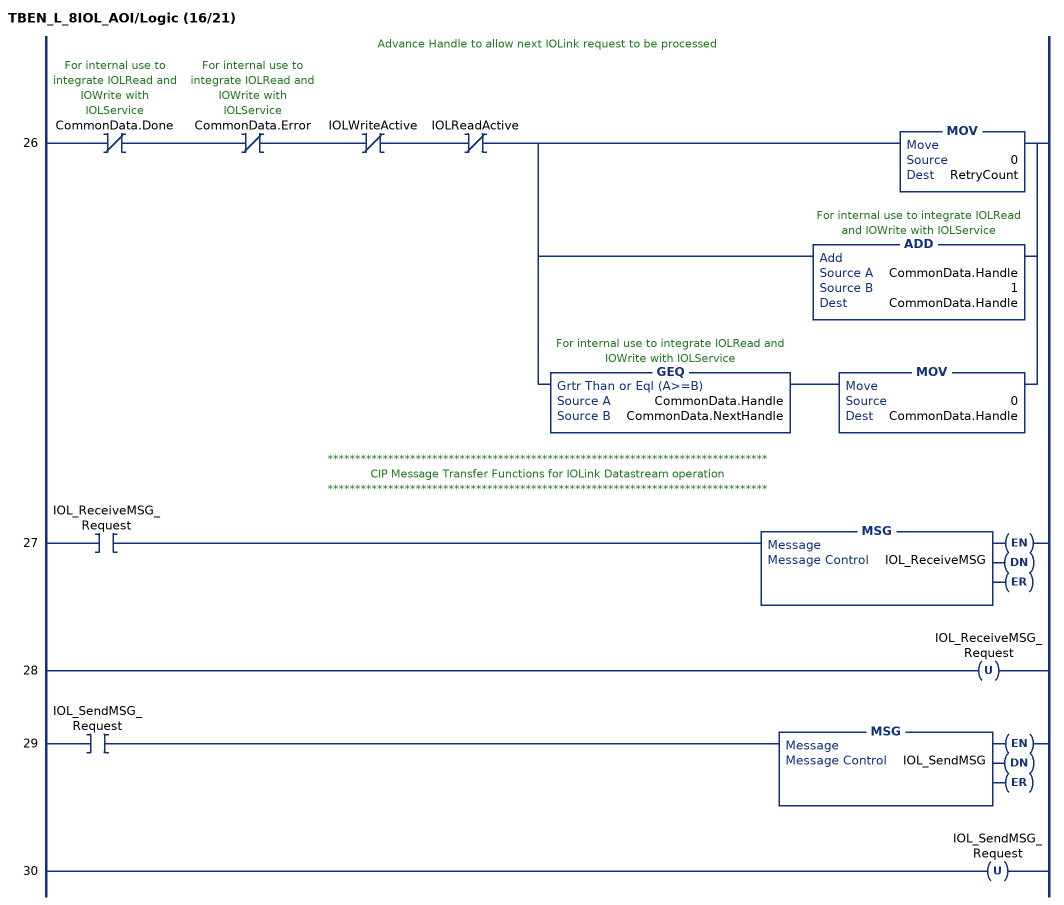
   // Advance Handle to allow next IOLink request to be processed
   26: XIO(CommonData.Done)XIO(CommonData.Error)XIO(IOLWriteActive)XIO(IOLReadActive)[MOV(0,RetryCount) ,ADD(CommonData.Handle,1,CommonData.Handle) ,GEQ(CommonData.Handle,CommonData.NextHandle) MOV(0,CommonData.Handle) ];
   // ********************************************************************************
   // CIP Message Transfer Functions for IOLink Datastream operation
   // ********************************************************************************
   27: XIC(IOL_ReceiveMSG_Request)MSG(IOL_ReceiveMSG);
   28: OTU(IOL_ReceiveMSG_Request);
   29: XIC(IOL_SendMSG_Request)MSG(IOL_SendMSG);
   30: OTU(IOL_SendMSG_Request);
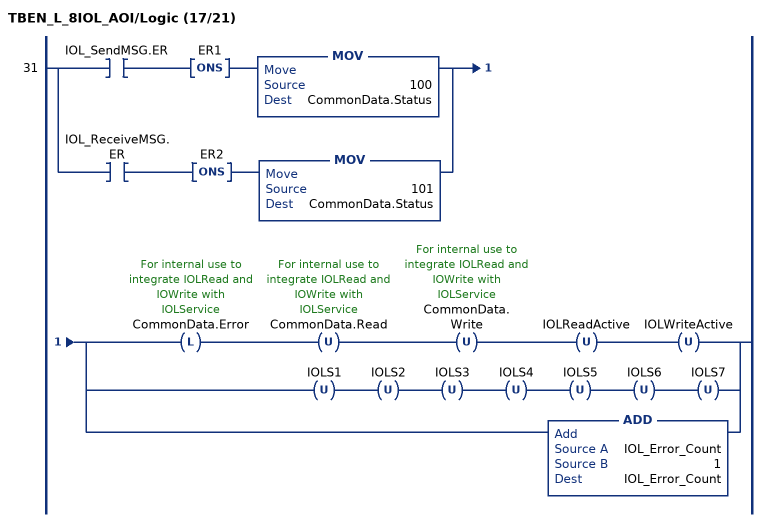
   31: [XIC(IOL_SendMSG.ER) ONS(ER1) MOV(100,CommonData.Status) ,XIC(IOL_ReceiveMSG.ER) ONS(ER2) MOV(101,CommonData.Status) ][OTL(CommonData.Error) OTU(CommonData.Read) OTU(CommonData.Write) OTU(IOLReadActive) OTU(IOLWriteActive) ,OTU(IOLS1) OTU(IOLS2) OTU(IOLS3) OTU(IOLS4) OTU(IOLS5) OTU(IOLS6) OTU(IOLS7) ,ADD(IOL_Error_Count,1,IOL_Error_Count) ];
